Staubli VAL3: onEditTrsf.pgx

public program onEditTrsf(num x_nIndex (dimensions=1), num x_nIndexItem (dimensions=1), string x_sEvent (dimensions=1))
  local num i
  local num l_nMin
  local num l_nMax
  local trsf l_tTrsf
  local string l_sEmpty
begin
  // edit TRSF OF THE POINT
  l_tTrsf=pEditPoint.tData[x_nIndexItem].pPoint.trsf
  // find the >
  call use:findPos(x_sEvent,">",i)
  i=i+1
  // find the line
  if !cycleStatus:bCycle
    l_nMin=l_nMax=0
  else
    switch x_nIndex
      case 0
        // x
        l_nMin=l_tTrsf.x-10
        l_nMax=l_tTrsf.x+10
      break
      case 1
        // y
        l_nMin=l_tTrsf.y-10
        l_nMax=l_tTrsf.y+10
      break
      case 2
        // z
        l_nMin=l_tTrsf.z-10
        l_nMax=l_tTrsf.z+10
      break
      case 3
        // rx
        l_nMin=l_tTrsf.rx-5
        l_nMax=l_tTrsf.rx+5
      break
      case 4
        // ry
        l_nMin=l_tTrsf.ry-5
        l_nMax=l_tTrsf.ry+5
      break
      case 5
        // rz
        l_nMin=l_tTrsf.rz-5
        l_nMax=l_tTrsf.rz+5
      break
    endSwitch
  endIf
  // clean the line
  call use:listcursor(use:nView,false)
  //
  switch x_nIndex
    case 0
      //  x-value
      call use:changeValue(l_tTrsf.x,l_nMin,l_nMax,i+40-use:nBottomX,use:nView+1,l_sEmpty)
    break
    case 1
      //  y-value
      call use:changeValue(l_tTrsf.y,l_nMin,l_nMax,i+40-use:nBottomX,use:nView+1,l_sEmpty)
    break
    case 2
      //  z-value
      call use:changeValue(l_tTrsf.z,l_nMin,l_nMax,i+40-use:nBottomX,use:nView+1,l_sEmpty)
    break
    case 3
      //  rx-value
      call use:changeValue(l_tTrsf.rx,l_nMin,l_nMax,i+40-use:nBottomX,use:nView+1,l_sEmpty)
    break
    case 4
      //  ry-value
      call use:changeValue(l_tTrsf.ry,l_nMin,l_nMax,i+40-use:nBottomX,use:nView+1,l_sEmpty)
    break
    case 5
      //  rz-value
      call use:changeValue(l_tTrsf.rz,l_nMin,l_nMax,i+40-use:nBottomX,use:nView+1,l_sEmpty)
    break
  endSwitch
  // validate
  if !use:bUseEscape
    pEditPoint.tData[x_nIndexItem].pPoint.trsf=l_tTrsf
  endIf
end
